// TIA Portal V19 export
TYPE "LUC_typeModeTransitionConfiguration"
// Configure in which states a mode transition is allowed
// stored: Access Published
   STRUCT
      clearing : Bool;   // Allow a mode transition to/from state Clearing
      stopped : Bool := true;   // Allow a mode transition to/from state Stopped
      starting : Bool;   // Allow a mode transition to/from state Starting
      idle : Bool := true;   // Allow a mode transition to/from state Idle
      suspended : Bool;   // Allow a mode transition to/from state Suspended
      execute : Bool;   // Allow a mode transition to/from state Execute
      stopping : Bool;   // Allow a mode transition to/from state Stopping
      aborting : Bool;   // Allow a mode transition to/from state Aborting
      aborted : Bool := true;   // Allow a mode transition to/from state Aborted
      holding : Bool;   // Allow a mode transition to/from state Holding
      held : Bool;   // Allow a mode transition to/from state Held
      unholding : Bool;   // Allow a mode transition to/from state Unholding
      suspending : Bool;   // Allow a mode transition to/from state Suspending
      unsuspending : Bool;   // Allow a mode transition to/from state Unsuspending
      resetting : Bool;   // Allow a mode transition to/from state Resetting
      completing : Bool;   // Allow a mode transition to/from state Completing
      completed : Bool;   // Allow a mode transition to/from state Completed
   END_STRUCT;
END_TYPE
